(* CoDeSys 2.3 export: STRUZSTATUS.EXP *)

(* Data type *)
(*Сигналы с част. преобр UZ*)
TYPE strUZStatus :
STRUCT
	Ready : BOOL;
	Running : BOOL;
	Fail	: BOOL;
END_STRUCT
END_TYPE
